(* IEC 61131-3 sources: dynamics/src, 28 files *)

(* ---- IDynamic.st ---- *)
NAMESPACE Dynamics
    INTERFACE IDynamic

        METHOD Next : LREAL
            VAR_INPUT
                value : LREAL;
            END_VAR
        END_METHOD

    END_INTERFACE
END_NAMESPACE

(* ---- IDynamicController.st ---- *)
NAMESPACE Dynamics
    INTERFACE IDynamicController

        METHOD Next : LREAL
            VAR_INPUT
                value : LREAL;
                input : LREAL;
            END_VAR
        END_METHOD

    END_INTERFACE
END_NAMESPACE

(* ---- IOutputDynamic.st ---- *)
NAMESPACE Simatic.Ax.Dynamics
    INTERFACE IOutputDynamic EXTENDS IDynamic, IOutputProvider
        METHOD SetOutput : LREAL
            VAR_INPUT
                output : LREAL;
            END_VAR
        END_METHOD
    END_INTERFACE
END_NAMESPACE

(* ---- IOutputProvider.st ---- *)
NAMESPACE Simatic.Ax.Dynamics
    INTERFACE IOutputProvider
        METHOD GetOutput : LREAL END_METHOD
    END_INTERFACE
END_NAMESPACE

(* ---- IOutputSignal.st ---- *)
NAMESPACE Dynamics
    INTERFACE IOutputSignal EXTENDS ISignal, IOutputProvider
    END_INTERFACE
END_NAMESPACE

(* ---- ISignal.st ---- *)
NAMESPACE Dynamics
    INTERFACE ISignal
        METHOD Next : LREAL END_METHOD
    END_INTERFACE
END_NAMESPACE

(* ---- Amplifier.st ---- *)
NAMESPACE Simatic.Ax.Dynamics
    CLASS Amplifier IMPLEMENTS IDynamic

        VAR PUBLIC
            k : LREAL := 1.0;
        END_VAR

        // Get K
        METHOD PUBLIC GetK : LREAL
            GetK := k;
        END_METHOD
        // Set K
        METHOD PUBLIC SetK
            VAR_INPUT
                newK : LREAL;
            END_VAR
            k := newK;
        END_METHOD

        METHOD PUBLIC Next : LREAL
            VAR_INPUT
                value : LREAL;
            END_VAR
            Next := k * value;
        END_METHOD

    END_CLASS
END_NAMESPACE

(* ---- BangBangController.st ---- *)
NAMESPACE Simatic.Ax.Dynamics
    CLASS BangBangController EXTENDS Controller

        VAR PUBLIC
            hysteresis : LREAL;
        END_VAR
        VAR PRIVATE
            _output : BOOL;
            _heatingMode : BOOL;
        END_VAR

        // Get Output
        METHOD PUBLIC GetOutput : BOOL
            GetOutput := _output;
        END_METHOD
        // Set Output
        METHOD PUBLIC SetOutput
            VAR_INPUT
                newOutput : BOOL;
            END_VAR
            _output := newOutput;
        END_METHOD

        // Get Mode
        METHOD PUBLIC IsHeatingModeEnabled : BOOL
            IsHeatingModeEnabled := _heatingMode;
        END_METHOD
        METHOD PUBLIC IsCoolingModeEnabled : BOOL
            IsCoolingModeEnabled := NOT _heatingMode;
        END_METHOD
        // Set Mode
        METHOD PUBLIC EnableHeatingMode
            _heatingMode := TRUE;
        END_METHOD
        METHOD PUBLIC EnableCoolingMode
            _heatingMode := FALSE;
        END_METHOD

        METHOD PUBLIC Next : BOOL
            VAR_INPUT
                value : LREAL;
            END_VAR
            IF      value < this.GetInput() - hysteresis THEN
                _output := _heatingMode;
            ELSIF   value > this.GetInput() + hysteresis THEN
                _output := NOT _heatingMode;
            END_IF;
            Next := _output;
        END_METHOD

        METHOD PUBLIC Next : BOOL
            VAR_INPUT
                value : LREAL;
                input : LREAL;
            END_VAR
            this.SetInput(input);
            Next := this.Next(value);
        END_METHOD

    END_CLASS
END_NAMESPACE

(* ---- BoundedDynamic.st ---- *)
NAMESPACE Simatic.Ax.Dynamics
    CLASS BoundedDynamic IMPLEMENTS IDynamic

        VAR PUBLIC
            unboundedDynamic : IDynamic;
            minOutput : LREAL;
            maxOutput : LREAL;
            observeMin : BOOL;
            observeMax : BOOL;
        END_VAR

        METHOD PUBLIC GetMinOutput : LREAL
            GetMinOutput := minOutput;
        END_METHOD
        METHOD PUBLIC SetMinOutput
            VAR_INPUT
                newMinOutput : LREAL;
            END_VAR
            observeMin := TRUE;
            minOutput := newMinOutput;
        END_METHOD
        METHOD PUBLIC DisableMin
            observeMin := FALSE;
        END_METHOD
        METHOD PUBLIC GetMaxOutput : LREAL
            GetMaxOutput := maxOutput;
        END_METHOD
        METHOD PUBLIC SetMaxOutput
            VAR_INPUT
                newMaxOutput : LREAL;
            END_VAR
            observeMax := TRUE;
            maxOutput := newMaxOutput;
        END_METHOD
        METHOD PUBLIC DisableMax
            observeMax := FALSE;
        END_METHOD

        METHOD PUBLIC Next : LREAL
            VAR_INPUT
                value : LREAL;
            END_VAR
            VAR_TEMP
                output : LREAL;
            END_VAR
            output := unboundedDynamic.Next(value);
            IF    observeMin AND output < minOutput THEN
                Next := minOutput;
            ELSIF observeMax AND output > maxOutput THEN
                Next := maxOutput;
            ELSE
                Next := output;
            END_IF;
        END_METHOD

    END_CLASS
END_NAMESPACE

(* ---- BoundedOutputDynamic.st ---- *)
NAMESPACE Dynamics
    CLASS BoundedOutputDynamic EXTENDS BoundedDynamic IMPLEMENTS IOutputDynamic

        VAR PRIVATE
            _storingDynamic : IOutputDynamic;
        END_VAR

        METHOD PUBLIC SetUnboundedDynamic
            VAR_INPUT
                newDynamic : IOutputDynamic;
            END_VAR
            _storingDynamic := newDynamic;
            unboundedDynamic := _storingDynamic;
        END_METHOD

        METHOD PUBLIC GetOutput : LREAL
            GetOutput := _storingDynamic.GetOutput();
        END_METHOD
        METHOD PUBLIC SetOutput : LREAL
            VAR_INPUT
                output : LREAL;
            END_VAR
            SetOutput := _storingDynamic.SetOutput(output);
        END_METHOD

        METHOD PUBLIC OVERRIDE Next : LREAL
            VAR_INPUT
                value : LREAL;
            END_VAR
            Next := _storingDynamic.SetOutput(SUPER.Next(value));
        END_METHOD

        METHOD PUBLIC IsMin : BOOL
            IsMin := _storingDynamic.GetOutput() = THIS.GetMinOutput();
        END_METHOD
        METHOD PUBLIC IsMax : BOOL
            IsMax := _storingDynamic.GetOutput() = THIS.GetMaxOutput();
        END_METHOD

    END_CLASS
END_NAMESPACE

(* ---- ConstantSignal.st ---- *)
NAMESPACE Simatic.Ax.Dynamics
    CLASS ConstantSignal IMPLEMENTS IOutputSignal

        VAR PUBLIC
            output : LREAL;
        END_VAR

        METHOD PUBLIC GetOutput : LREAL
            GetOutput := output;
        END_METHOD
        METHOD PUBLIC SetOutput : LREAL
            VAR_INPUT
                newOutput : LREAL;
            END_VAR
            output := newOutput;
            SetOutput := output;
        END_METHOD

        METHOD PUBLIC Next : LREAL
            Next := THIS.GetOutput();
        END_METHOD

    END_CLASS
END_NAMESPACE

(* ---- ConstantTimeProvider.st ---- *)
NAMESPACE TimeProviders
    CLASS ConstantTimeProvider IMPLEMENTS IElapsedSecondsProvider

        VAR PUBLIC
            seconds : LREAL;
        END_VAR

        METHOD PUBLIC GetElapsedSeconds : LREAL
            GetElapsedSeconds := seconds;
        END_METHOD

        METHOD PUBLIC Start
            ; // Nothing happens -- that's why it's called constant
        END_METHOD

END_CLASS
END_NAMESPACE

(* ---- Controller.st ---- *)
NAMESPACE Simatic.Ax.Dynamics
    CLASS INTERNAL Controller

        VAR PRIVATE
            _input : LREAL;
        END_VAR

        METHOD PUBLIC GetInput : LREAL
            GetInput := _input;
        END_METHOD
        METHOD PUBLIC SetInput
            VAR_INPUT
                newInput : LREAL;
            END_VAR
            _input := newInput;
        END_METHOD

    END_CLASS
END_NAMESPACE

(* ---- Differentiator.st ---- *)
NAMESPACE Dynamics
    CLASS Differentiator EXTENDS FirstOrderDynamic

        VAR PUBLIC
            tDSeconds : LREAL;
        END_VAR

        VAR PRIVATE
            _value : LREAL;
        END_VAR

        METHOD PUBLIC GetTDSeconds : LREAL
            GetTDSeconds := tDSeconds;
        END_METHOD
        METHOD PUBLIC SetTDSeconds
            VAR_INPUT
                newTDSeconds : LREAL;
            END_VAR
            tDSeconds := newTDSeconds;
        END_METHOD
        METHOD PUBLIC SetTDSeconds
            VAR_INPUT
                newTDSeconds : LREAL;
                k : LREAL;
            END_VAR
            THIS.SetTDSeconds(newTDSeconds * k);
        END_METHOD

        METHOD INTERNAL GetValue : LREAL
            GetValue := _value;
        END_METHOD

        METHOD PROTECTED OVERRIDE _Next : LREAL
            VAR_INPUT
                value : LREAL;
                elapsedSeconds : LREAL;
            END_VAR
            _Next := (value - _value) / elapsedSeconds * tDSeconds;
            _value := value;
        END_METHOD

    END_CLASS
END_NAMESPACE

(* ---- DynamicController.st ---- *)
NAMESPACE Simatic.Ax.Dynamics
    CLASS DynamicController EXTENDS Controller IMPLEMENTS IDynamic, IDynamicController

        VAR PUBLIC
            openDynamic : IDynamic;
        END_VAR

        METHOD PUBLIC Next : LREAL
            VAR_INPUT
                value : LREAL;
            END_VAR
            Next := openDynamic.Next(THIS.GetInput() - value);
        END_METHOD

        METHOD PUBLIC Next : LREAL
            VAR_INPUT
                value : LREAL;
                input : LREAL;
            END_VAR
            THIS.SetInput(input);
            Next := THIS.Next(value);
        END_METHOD

    END_CLASS
END_NAMESPACE

(* ---- ExplicitSignal.st ---- *)
NAMESPACE Dynamics
    CLASS ABSTRACT ExplicitSignal IMPLEMENTS IOutputSignal

        VAR PRIVATE
            _cycle : UINT;
        END_VAR

        METHOD PUBLIC Reset
            _cycle := UINT#0;
        END_METHOD

        METHOD PROTECTED ABSTRACT _GetOutput : LREAL
            VAR_INPUT
                cycle : UINT;
            END_VAR
        END_METHOD

        METHOD PUBLIC FINAL GetOutput : LREAL
            GetOutput := THIS._GetOutput(_cycle);
        END_METHOD

        METHOD PUBLIC FINAL Next : LREAL
            _cycle := _cycle + UINT#1;
            Next := THIS.GetOutput();
        END_METHOD

    END_CLASS
END_NAMESPACE

(* ---- FirstOrderDynamic.st ---- *)
USING TimeProviders;
NAMESPACE Simatic.Ax.Dynamics
    CLASS INTERNAL ABSTRACT FirstOrderDynamic IMPLEMENTS IDynamic

        VAR PUBLIC
            elapsedTimeProvider : IElapsedSecondsProvider;
        END_VAR

        METHOD PROTECTED ABSTRACT _Next : LREAL
            VAR_INPUT
                value : LREAL;
                elapsedSeconds : LREAL;
            END_VAR
        END_METHOD
        METHOD PUBLIC FINAL Next : LREAL
            VAR_INPUT
                value : LREAL;
            END_VAR
            Next := this._Next(value, elapsedTimeProvider.GetElapsedSeconds());
            elapsedTimeProvider.Start();
        END_METHOD

    END_CLASS
END_NAMESPACE

(* ---- FirstOrderOutputDynamic.st ---- *)
NAMESPACE Dynamics
    CLASS INTERNAL ABSTRACT FirstOrderOutputDynamic EXTENDS FirstOrderDynamic IMPLEMENTS IOutputDynamic

        VAR PRIVATE
            _output : LREAL;
        END_VAR

        METHOD PUBLIC GetOutput : LREAL
            GetOutput := _output;
        END_METHOD
        METHOD PUBLIC SetOutput : LREAL
            VAR_INPUT
                output : LREAL;
            END_VAR
            _output := output;
            SetOutput := _output;
        END_METHOD

        METHOD PROTECTED ABSTRACT _Next : LREAL
            VAR_INPUT
                value : LREAL;
                elapsedSeconds : LREAL;
                output : LREAL;
            END_VAR
        END_METHOD

        METHOD PROTECTED FINAL OVERRIDE _Next : LREAL
            VAR_INPUT
                value : LREAL;
                elapsedSeconds : LREAL;
            END_VAR
            _Next := this.SetOutput(this._Next(value, elapsedSeconds, _output));
        END_METHOD

    END_CLASS
END_NAMESPACE

(* ---- IdentityDynamic.st ---- *)
NAMESPACE Dynamics
    CLASS IdentityDynamic IMPLEMENTS IDynamic

        METHOD PUBLIC Next : LREAL
            VAR_INPUT
                value : LREAL;
            END_VAR
            Next := value;
        END_METHOD

    END_CLASS
END_NAMESPACE

(* ---- Integrator.st ---- *)
NAMESPACE Simatic.Ax.Dynamics
    CLASS Integrator EXTENDS FirstOrderOutputDynamic

        VAR PUBLIC
            tISeconds : LREAL;
        END_VAR

        METHOD PUBLIC GetTISeconds : LREAL
            GetTISeconds := tISeconds;
        END_METHOD
        METHOD PUBLIC SetTISeconds
            VAR_INPUT
                newTISeconds : LREAL;
            END_VAR
            tISeconds := newTISeconds;
        END_METHOD
        METHOD PUBLIC SetTISeconds
            VAR_INPUT
                newTISeconds : LREAL;
                k : LREAL;
            END_VAR
            THIS.SetTISeconds(newTISeconds / k);
        END_METHOD

        METHOD PROTECTED OVERRIDE _Next : LREAL
            VAR_INPUT
                value : LREAL;
                elapsedSeconds : LREAL;
                output : LREAL;
            END_VAR
            _Next := output + value * elapsedSeconds / tISeconds;
        END_METHOD

    END_CLASS
END_NAMESPACE

(* ---- myClass.st ---- *)
NAMESPACE Simatic.Ax.Library

    {axcode:docs-v0:@simatic-ax/dynamics:MyClass.md}
    CLASS MyClass

        VAR PUBLIC
        END_VAR

        VAR
        END_VAR

        /// Inline Comment for MyMethod. It will be shown, when you hover over the method
        /// This method has no parameters and no return value
        METHOD PUBLIC MyMethod
            ;
        END_METHOD

    END_CLASS

END_NAMESPACE

(* ---- ParallelFirstOrderDynamic.st ---- *)
USING TimeProviders;
USING TimeProviders;
NAMESPACE Simatic.Ax.Dynamics
    CLASS INTERNAL ABSTRACT ParallelFirstOrderDynamic EXTENDS FirstOrderDynamic

        VAR PUBLIC
            k : LREAL := 1.0;
        END_VAR

        VAR PROTECTED
            _pseudoTimeProvider : ConstantTimeProvider;
        END_VAR

        METHOD PUBLIC GetK : LREAL
            GetK := k;
        END_METHOD
        METHOD PUBLIC SetK
            VAR_INPUT
                newK : LREAL;
            END_VAR
            k := newK;
        END_METHOD

        METHOD PROTECTED ABSTRACT _Next0 : LREAL
            VAR_INPUT
                value : LREAL;
            END_VAR
        END_METHOD
        METHOD PROTECTED ABSTRACT _Next1 : LREAL
            VAR_INPUT
                value : LREAL;
            END_VAR
        END_METHOD

        METHOD PROTECTED FINAL OVERRIDE _Next : LREAL
            VAR_INPUT
                value : LREAL;
                elapsedSeconds : LREAL;
            END_VAR
            _pseudoTimeProvider.seconds := elapsedSeconds;
            _Next := k * (this._Next0(value) + this._Next1(value));
        END_METHOD

    END_CLASS
END_NAMESPACE

(* ---- PD_Dynamic.st ---- *)
NAMESPACE Simatic.Ax.Dynamics
    CLASS PD_Dynamic EXTENDS ParallelFirstOrderDynamic

        VAR PRIVATE
            _differentiator : Differentiator;
        END_VAR

        METHOD PUBLIC GetTDSeconds : LREAL
            GetTDSeconds := _differentiator.GetTDSeconds();
        END_METHOD
        METHOD PUBLIC SetTDSeconds
            VAR_INPUT
                newTDSeconds : LREAL;
            END_VAR
            _differentiator.SetTDSeconds(newTDSeconds);
            _differentiator.elapsedTimeProvider := _pseudoTimeProvider;
        END_METHOD

        // P
        METHOD PROTECTED OVERRIDE _Next0 : LREAL
            VAR_INPUT
                value : LREAL;
            END_VAR
            _Next0 := value;
        END_METHOD

        // D
        METHOD PROTECTED OVERRIDE _Next1 : LREAL
            VAR_INPUT
                value : LREAL;
            END_VAR
            _Next1 := _differentiator.Next(value);
        END_METHOD

    END_CLASS
END_NAMESPACE

(* ---- PI_Dynamic.st ---- *)
NAMESPACE Simatic.Ax.Dynamics
    CLASS PI_Dynamic EXTENDS ParallelFirstOrderDynamic

        VAR PRIVATE
            _boundedIntegrator : BoundedOutputDynamic;
            _unboundedIntegrator : Integrator;
        END_VAR

        METHOD PUBLIC GetTISeconds : LREAL
            GetTISeconds := _unboundedIntegrator.GetTISeconds();
        END_METHOD
        METHOD PUBLIC SetTISeconds : LREAL
            VAR_INPUT
                seconds : LREAL;
            END_VAR
            _boundedIntegrator.SetUnboundedDynamic(_unboundedIntegrator);
            _unboundedIntegrator.elapsedTimeProvider := _pseudoTimeProvider;
            _unboundedIntegrator.SetTISeconds(seconds);
        END_METHOD

        METHOD PUBLIC GetIntegratorMinOutput : LREAL
            GetIntegratorMinOutput := _boundedIntegrator.GetMinOutput();
        END_METHOD
        METHOD PUBLIC SetIntegratorMinOutput : LREAL
            VAR_INPUT
                newMinOutput : LREAL;
            END_VAR
            _boundedIntegrator.SetMinOutput(newMinOutput);
        END_METHOD
        METHOD PUBLIC DisableIntegratorMin
            _boundedIntegrator.DisableMin();
        END_METHOD
        METHOD PUBLIC GetIntegratorMaxOutput : LREAL
            GetIntegratorMaxOutput := _boundedIntegrator.GetMaxOutput();
        END_METHOD
        METHOD PUBLIC SetIntegratorMaxOutput : LREAL
            VAR_INPUT
                newMaxOutput : LREAL;
            END_VAR
            _boundedIntegrator.SetMaxOutput(newMaxOutput);
        END_METHOD
        METHOD PUBLIC DisableIntegratorMax
            _boundedIntegrator.DisableMax();
        END_METHOD

        // P
        METHOD PROTECTED OVERRIDE _Next0 : LREAL
            VAR_INPUT
                value : LREAL;
            END_VAR
            _Next0 := value;
        END_METHOD

        // I
        METHOD PROTECTED OVERRIDE _Next1 : LREAL
            VAR_INPUT
                value : LREAL;
            END_VAR
            _Next1 := _boundedIntegrator.Next(value);
        END_METHOD
    END_CLASS
END_NAMESPACE

(* ---- PID_Dynamic.st ---- *)
NAMESPACE Simatic.Ax.Dynamics
    CLASS PID_Dynamic EXTENDS ParallelFirstOrderDynamic

        VAR PRIVATE
            _pi_dynamic : PI_Dynamic;
            _d_dynamic : Differentiator;
        END_VAR

        // Get TI
        METHOD PUBLIC GetTISeconds : LREAL
            GetTISeconds := _pi_dynamic.GetTISeconds();
        END_METHOD
        //Set TI
        METHOD PUBLIC SetTISeconds : LREAL
            VAR_INPUT
                seconds : LREAL;
            END_VAR
            _pi_dynamic.SetTISeconds(seconds);
            _pi_dynamic.elapsedTimeProvider := _pseudoTimeProvider;
        END_METHOD

        // Get TD
        METHOD PUBLIC GetTDSeconds : LREAL
            GetTDSeconds := _d_dynamic.GetTDSeconds();
        END_METHOD
        // Set TD
        METHOD PUBLIC SetTDSeconds
            VAR_INPUT
                newTDSeconds : LREAL;
            END_VAR
            _d_dynamic.SetTDSeconds(newTDSeconds);
            _d_dynamic.elapsedTimeProvider := _pseudoTimeProvider;
        END_METHOD

        METHOD PUBLIC GetIntegratorMinOutput : LREAL
            GetIntegratorMinOutput := _pi_dynamic.GetIntegratorMinOutput();
        END_METHOD
        METHOD PUBLIC SetIntegratorMinOutput : LREAL
            VAR_INPUT
                newMinOutput : LREAL;
            END_VAR
            _pi_dynamic.SetIntegratorMinOutput(newMinOutput);
        END_METHOD
        METHOD PUBLIC GetIntegratorMaxOutput : LREAL
            GetIntegratorMaxOutput := _pi_dynamic.GetIntegratorMaxOutput();
        END_METHOD
        METHOD PUBLIC SetIntegratorMaxOutput : LREAL
            VAR_INPUT
                newMaxOutput : LREAL;
            END_VAR
            _pi_dynamic.SetIntegratorMaxOutput(newMaxOutput);
        END_METHOD

        // PI
        METHOD PROTECTED OVERRIDE _Next0 : LREAL
            VAR_INPUT
                value : LREAL;
            END_VAR
            _Next0 := _pi_dynamic.Next(value);
        END_METHOD

        // D
        METHOD PROTECTED OVERRIDE _Next1 : LREAL
            VAR_INPUT
                value : LREAL;
            END_VAR
            _Next1 := _d_dynamic.Next(value);
        END_METHOD
    END_CLASS
END_NAMESPACE

(* ---- PT1_DeadbeatController.st ---- *)
USING System.Math;
NAMESPACE Dynamics
    CLASS PT1_DeadbeatController EXTENDS Controller IMPLEMENTS IDynamicController

        VAR PROTECTED
            _expTT : LREAL;
            _k : LREAL;
        END_VAR

        // Get K
        METHOD PUBLIC GetK : LREAL
            GetK := _k;
        END_METHOD
        // Set K
        METHOD PUBLIC SetK
            VAR_INPUT
                k : LREAL;
            END_VAR
            _k := k;
        END_METHOD

        // Set T0
        METHOD PUBLIC SetPeriods
            VAR_INPUT
                elapsedTime : LREAL;
                t0 : LREAL;
            END_VAR
            _expTT := Exp(elapsedTime / t0);
        END_METHOD

        METHOD PUBLIC Next : LREAL
            VAR_INPUT
                value : LREAL;
            END_VAR
            Next := (THIS.GetInput() * _expTT - value) / (_expTT - 1) / _k;
        END_METHOD

        METHOD PUBLIC Next : LREAL
            VAR_INPUT
                value : LREAL;
                input : LREAL;
            END_VAR
            THIS.SetInput(input);
            Next := THIS.Next(value);
        END_METHOD

    END_CLASS
END_NAMESPACE

(* ---- PT1_Dynamic.st ---- *)
NAMESPACE Simatic.Ax.Dynamics
    CLASS PT1_Dynamic EXTENDS FirstOrderOutputDynamic

        VAR PUBLIC
            k : LREAL;
            t0Seconds : LREAL;
        END_VAR

        METHOD PUBLIC GetK : LREAL
            GetK := k;
        END_METHOD
        METHOD PUBLIC SetK
            VAR_INPUT
                newK : LREAL;
            END_VAR
            k := newK;
        END_METHOD

        METHOD PUBLIC GetT0Seconds : LREAL
            GetT0Seconds := t0Seconds;
        END_METHOD
        METHOD PUBLIC SetT0Seconds
            VAR_INPUT
                newT0Seconds : LREAL;
            END_VAR
            t0Seconds := newT0Seconds;
        END_METHOD

        METHOD PROTECTED OVERRIDE _Next : LREAL
            VAR_INPUT
                value : LREAL;
                elapsedSeconds : LREAL;
                output : LREAL;
            END_VAR
            _Next := output + (k * value - output) * elapsedSeconds / t0Seconds;
        END_METHOD

    END_CLASS
END_NAMESPACE

(* ---- RampSignal.st ---- *)
NAMESPACE Simatic.Ax.Dynamics
    CLASS RampSignal IMPLEMENTS IOutputSignal

        VAR PUBLIC
            elapsedTimeProvider : TimeProviders.IElapsedSecondsProvider;
            slope : LREAL;
        END_VAR
        VAR PRIVATE
            _output : LREAL;
        END_VAR

        // Get output
        METHOD PUBLIC GetOutput : LREAL
            GetOutput := _output;
        END_METHOD
        // Set output
        METHOD PUBLIC SetOutput : LREAL
            VAR_INPUT
                newOutput : LREAL;
            END_VAR
            _output := newOutput;
            SetOutput := _output;
        END_METHOD

        METHOD PUBLIC  GetTISeconds : LREAL
            GetTISeconds := 1 / slope;
        END_METHOD
        METHOD PUBLIC SetTISeconds
            VAR_INPUT
                newTISeconds : LREAL;
            END_VAR
            slope := 1 / newTISeconds;
        END_METHOD

        METHOD PUBLIC Next : LREAL
            _output := _output + elapsedTimeProvider.GetElapsedSeconds() * slope;
            Next := _output;
        END_METHOD

    END_CLASS
END_NAMESPACE
